TYPE E_TL_Sensors :
(
	eCounterSensor := 1,
	eTlMaxNumSensors
)UINT;
END_TYPE

(* stored: Version 1.1.0.1, ProductVersion 3.1.4024.0
   DUT E_TL_Sensors: Id {fba731ae-a66e-47a4-9c19-af5c6ec300dd} *)
